{attribute 'qualified_only'}
{attribute 'strict'}
{attribute 'to_string'}
TYPE E_MESSAGE_CHECK :
(
  NULL,
  // 9000 --> here comes your error
  POINTER_INVALID             := 9000,
  POINTER_TIME_INVALID,
  POINTER_LIST_INVALID,
  POINTER_MSG_IDX_INVALID,
  POINTER_ERR_IDX_INVALID,
  POINTER_ROOT_FILE_INVALID,
  POINTER_ROOT_DIR_INVALID,
  POINTER_CTRL_INVALID,
  POINTER_STATE_INVALID,

  // 10000 --> here comes your man
  CHECK_DONE                        := 10000
)UINT;
END_TYPE

(* stored: Version 1.1.0.1, ProductVersion 3.1.4026.18
   DUT E_MESSAGE_CHECK: Id {f1b81a6c-f378-4de9-bdd1-64f881b40300} *)
